Yaskawa INFORM job: �l�.JBI

/JOB
//NAME 俵倝倢倧
//POS
///NPOS 5,0,0,0
///TOOL 0
///PULSE
C000=-2,0,292,-1,0,-1
C001=-2,30672,-29900,-1,0,-1
C002=-2,30672,-29900,4535,0,2211
C003=-2,30672,-29900,-3837,0,-2689
C004=-2,52752,-56492,-3837,0,-2689
//INST
///DATE 2014/09/13 20:51
///ATTR 0,0,0,0,0,0,0,0,0,0,0,0,0,1,0,0
///FRAME BASE
NOP
*L
MOVJ C000 VJ=50.00 CONT
MOVJ C001 VJ=100.00 CONT
MOVJ C002 VJ=100.00 CONT
MOVJ C003 VJ=100.00 CONT
MOVJ C004 VJ=60.00 CONT
JUMP *L
END
